PROGRAM pouS2Warnings
VAR
	
idbMsgWarn: FB_CheckMessageBounds;
END_VAR

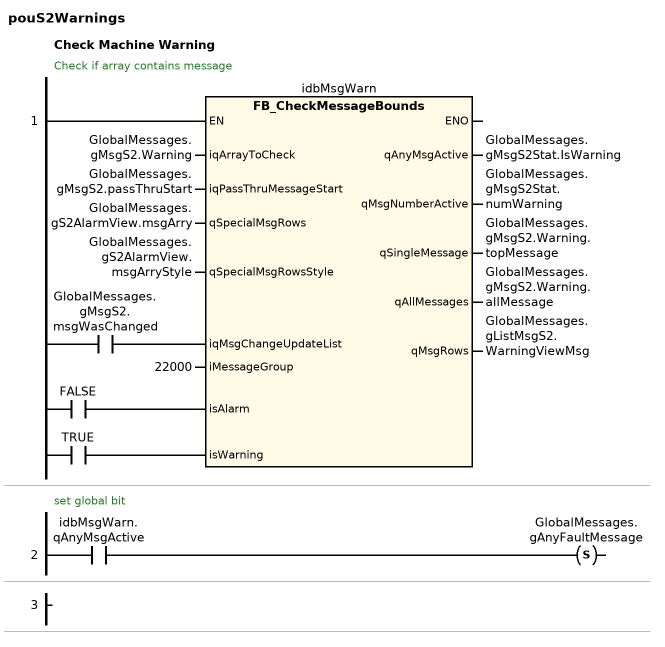
// NETWORK 1: Check Machine Warning
// Check if array contains message
idbMsgWarn(
    iqArrayToCheck := GlobalMessages.gMsgS2.Warning,
    iqPassThruMessageStart := GlobalMessages.gMsgS2.passThruStart,
    qSpecialMsgRows := GlobalMessages.gS2AlarmView.msgArry,
    qSpecialMsgRowsStyle := GlobalMessages.gS2AlarmView.msgArryStyle,
    iqMsgChangeUpdateList := GlobalMessages.gMsgS2.msgWasChanged,
    iMessageGroup := 22000,
    isAlarm := FALSE,
    isWarning := TRUE,
    qAnyMsgActive => GlobalMessages.gMsgS2Stat.IsWarning,
    qMsgNumberActive => GlobalMessages.gMsgS2Stat.numWarning,
    qSingleMessage => GlobalMessages.gMsgS2.Warning.topMessage,
    qAllMessages => GlobalMessages.gMsgS2.Warning.allMessage,
    qMsgRows => GlobalMessages.gListMsgS2.WarningViewMsg); // FB_CheckMessageBounds

// NETWORK 2
// set global bit
GlobalMessages.gAnyFaultMessage S= idbMsgWarn.qAnyMsgActive;

// NETWORK 3

END_PROGRAM

(* stored: Version 1.1.0.1, ProductVersion 3.1.4024.12
   POU pouS2Warnings: Id {59e492b6-a3ee-4ea8-9703-5170e9b15f2c}, SpecialFunc None *)
